FUNCTION_BLOCK ABSTRACT SuspendedProgramState EXTENDS ProgramState

{attribute 'monitoring' := 'call'}
{attribute 'OPC.UA.DA.Property' := '1'}
{attribute 'OPC.UA.DA.Access' := '1'}
PROPERTY FINAL Name : STRING
GET
Name := 'Suspended';
END_GET
END_PROPERTY

END_FUNCTION_BLOCK

(* stored: Version 1.1.0.1
   POU SuspendedProgramState: Id {44690efb-abcd-486a-acbb-08acdab2a352}, SpecialFunc None
   Property Name: Id {930130f5-7e88-4946-8fab-d91419aa18d5}
   Get Get: Id {e232729c-09b7-491b-9a90-95bb9852b556} *)
